// TwinCAT 3 PLC project
// project tree:
//   POUs/ func_f.TcPOU, normProjIdx.TcPOU (not stored), MAIN.TcPOU, makeArray0.TcPOU, makeTupleStruct_1.TcPOU (not stored), proj0_TupleStruct_1.TcPOU (not stored), proj1_TupleStruct_1.TcPOU (not stored)
//   DUTs/ STATE.TcDUT, TupleStruct_1.TcDUT (not stored)
//   GVLs/ INPUTS.TcGVL, TIMERS.TcGVL (not stored)

// ---- DUTs/STATE.TcDUT
TYPE STATE:
    STRUCT
        curTime: LREAL;
        dvar_M_a_li AT %Q*: ARRAY[0..4] of DINT;
    END_STRUCT
END_TYPE

// ---- GVLs/INPUTS.TcGVL
VAR_GLOBAL // INPUTS
    ivar_i AT %I*: BOOL;
END_VAR

// ---- POUs/func_f.TcPOU
FUNCTION func_f: DINT
VAR_INPUT
    farg2_f_p: ARRAY[0..4] of DINT;
END_VAR
VAR
    farg_f_p: ARRAY[0..4] of DINT;
END_VAR

farg_f_p := farg2_f_p;
farg_f_p[normProjIdx(0, 5)] := 5;
farg_f_p[normProjIdx(1, 5)] := 6;
func_f := ((((farg_f_p[normProjIdx(0, 5)]) + (farg_f_p[normProjIdx(1, 5)])) + (farg_f_p[normProjIdx(2, 5)])) + (farg_f_p[normProjIdx(3, 5)])) + (farg_f_p[normProjIdx(4, 5)]);
RETURN;

END_FUNCTION

// ---- POUs/MAIN.TcPOU

      PROGRAM MAIN
VAR_OUTPUT
    timerValue0: TIME;
    timerValue1: TIME;
END_VAR
VAR
    cnt: LINT;
    first: BOOL := TRUE;
    curTimerValue: TIME;
    state0: STATE;
    curTime: LREAL;
    loopsKilled: LINT;
END_VAR
VAR_TEMP
    lastTimerValue: TIME;
    curDeltaTime: TIME;
    curDeltaSecs: LREAL;
    state1: STATE;
    progress: BOOL;
    loopCount: INT;
END_VAR


        
// Handle 'time' and cycle time.
cnt := cnt + 1;

timer0(IN := curTimer = 0, PT := T#1D);
timer1(IN := curTimer = 1, PT := T#1D);
timerValue0 := timer0.ET;
timerValue1 := timer1.ET;

lastTimerValue := curTimerValue;
IF curTimer = 0 THEN
    curTimerValue := timerValue0;
ELSE
    curTimerValue := timerValue1;
END_IF;
curDeltaTime := curTimerValue - lastTimerValue;
curDeltaSecs := TIME_TO_LREAL(curDeltaTime) / 1000;
curTime := curTime + curDeltaSecs;

IF cnt MOD 10 = 0 THEN
    curTimer := 1 - curTimer;
    curTimerValue := T#0S;
    timer0(IN := curTimer = 0, PT := T#1D);
    timer1(IN := curTimer = 1, PT := T#1D);
    timerValue0 := timer0.ET;
    timerValue1 := timer1.ET;
END_IF;

IF first THEN
    first := FALSE;

    // Initialize state variables for initial state.
    state0.dvar_M_a_li := makeArray0(0, 0, 0, 0, 0);
ELSE
    // Update continuous variables for time delay.

    state0.curTime := curTime;
END_IF;

// Event loop.
WHILE TRUE DO
    progress := FALSE;

    // Event "tau".
    IF NOT progress THEN
        IF (func_f(state0.dvar_M_a_li)) = (9) THEN
            progress := TRUE;
            state1 := state0;

            state1.dvar_M_a_li[normProjIdx(0, 5)] := 5;
            state1.dvar_M_a_li[normProjIdx(1, 5)] := 6;

            state0 := state1;
        END_IF;
    END_IF;

    // Event "tau".
    IF NOT progress THEN
        IF (func_f(state0.dvar_M_a_li)) = (10) THEN
            progress := TRUE;
            state1 := state0;

            state1.dvar_M_a_li[normProjIdx(2, 5)] := proj0_TupleStruct_1(makeTupleStruct_1(7, 8));
            state1.dvar_M_a_li[normProjIdx(3, 5)] := proj1_TupleStruct_1(makeTupleStruct_1(7, 8));

            state0 := state1;
        END_IF;
    END_IF;

    // Done with events?
    IF NOT progress THEN
        EXIT;
    END_IF;

    // Protect against events that are always enabled.
    loopCount := loopCount + 1;
    IF loopCount >= 100 THEN
        loopsKilled := loopsKilled + 1;
        EXIT;
    END_IF;
END_WHILE;

END_PROGRAM

// ---- POUs/makeArray0.TcPOU

      FUNCTION makeArray0: ARRAY[0..4] of DINT
VAR_INPUT
    elem0: DINT;
    elem1: DINT;
    elem2: DINT;
    elem3: DINT;
    elem4: DINT;
END_VAR
VAR
    rslt: ARRAY[0..4] of DINT;
END_VAR


        rslt[0] := elem0;
rslt[1] := elem1;
rslt[2] := elem2;
rslt[3] := elem3;
rslt[4] := elem4;
makeArray0 := rslt;

END_FUNCTION
